TYPE E_EmulatedState :
(
	StaticData := 0,
	SimulinkPlant,
	VirtualPlant,
	PhysicalPlant	
) DINT;
END_TYPE

(* stored: Version 1.1.0.1, ProductVersion 3.1.4022.11
   DUT E_EmulatedState: Id {20e3c706-d939-462e-877b-84c60541d5f7} *)
